TYPE EM_Transport_HMI :
STRUCT
	Start		: BOOL;
	Stop		: BOOL;
	Reset		: BOOL;
	Abort		: BOOL;
	Auto		: BOOL;
	Manueel		: BOOL;
	Clear		: BOOL;
	UnSuspend	: BOOL;
	Suspend		: BOOL;
	UnHold		: BOOL;
	Hold		: BOOL;
END_STRUCT
END_TYPE

(* stored: Version 1.1.0.1, ProductVersion 3.1.4024.12
   DUT EM_Transport_HMI: Id {aed052bd-58c1-4577-9e04-db27ab8dcd0d} *)
